/// Monitor enabled work areas
FUNCTION_BLOCK MonitorWorkAreaFB EXTENDS RobotLibraryBaseFB
// ------------------------------------------------------------------------- 
//  SRCI Robot Library                                                
// ------------------------------------------------------------------------- 
//                                                                           
//  Object:      MonitorWorkAreaFB                                       
//  Author:      Thorsten Brach                                                
//  Date:        2024-06-01
//
//  Description:                                              
//   
//                                                                           
//  Copyright: 
//    (C) 2024 Thorsten Brach. All rights reserved                                                                         
//                                                                           
//  Disclaimer:                                                                           
//    This project is provided without any guarantee and can be used for   
//    private and commercial purposes. Any commercial use is at the user’s 
//    own risk and responsibility.
//
// -------------------------------------------------------------------------
VAR_INPUT
  /// Start of the command at the rising edge
  Execute            : BOOL;
  /// Index of robot work area to be monitored
  /// • 0 (default)..254
  WorkAreaNo         : USINT;
END_VAR

VAR_OUTPUT
  /// TRUE, while the following outputs return valid values
  /// ActivationState
  /// MonitoringState
  Valid              : BOOL;
  /// FB is being processed
  Busy               : BOOL;
  /// Command is transferred and confirmed by the RC
  CommandBuffered    : BOOL;  
  /// Receiving of input parameter values has been acknowledged by RC
  ParameterAccepted  : BOOL;
  /// Bits return TRUE when work area defined by Index is active
  ActivationState    : WORD;
  /// Bits return TRUE when violation is reported.
  MonitoringState    : WORD;
END_VAR

                  
                

METHOD PROTECTED OnCall
VAR_IN_OUT
  /// Robot assignment of function
  AxesGroup         : AxesGroup; 
END_VAR
                        
                      
END_METHOD
END_FUNCTION_BLOCK

/// Switch path mode between high and low accuracy
FUNCTION_BLOCK PathAccuracyModeFB EXTENDS RobotLibraryBaseFB
// ------------------------------------------------------------------------- 
//  SRCI Robot Library                                                
// ------------------------------------------------------------------------- 
//                                                                           
//  Object:      PathAccuracyModeFB                                       
//  Author:      Thorsten Brach                                                
//  Date:        2024-06-01
//
//  Description:                                              
//   
//                                                                           
//  Copyright: 
//    (C) 2024 Thorsten Brach. All rights reserved                                                                         
//                                                                           
//  Disclaimer:                                                                           
//    This project is provided without any guarantee and can be used for   
//    private and commercial purposes. Any commercial use is at the user’s 
//    own risk and responsibility.
//
// -------------------------------------------------------------------------
VAR_INPUT
  /// Set TRUE to change RA power state to "Enabled"
  Enable            : BOOL;
END_VAR

VAR_OUTPUT
  /// FB is being processed
  Busy              : BOOL;
  /// Command is transferred and confirmed by the RC
  CommandBuffered   : BOOL;
  /// TRUE while PathAccuracyMode is active
  Enabled           : BOOL;
  /// Receiving of input parameter values has been acknowledged by RC
  ParameterAccepted : BOOL;
END_VAR

                  
                

METHOD PROTECTED OnCall
VAR_IN_OUT
  /// Robot assignment of function
  AxesGroup         : AxesGroup; 
END_VAR
                        
                      
END_METHOD
END_FUNCTION_BLOCK

/// Restart/reboot of the RC.
FUNCTION_BLOCK RestartControllerFB EXTENDS RobotLibraryBaseFB
// ------------------------------------------------------------------------- 
//  SRCI Robot Library                                                
// ------------------------------------------------------------------------- 
//                                                                           
//  Object:      RestartControllerFB                                       
//  Author:      Thorsten Brach                                                
//  Date:        2024-06-01
//
//  Description:                                              
//   
//                                                                           
//  Copyright: 
//    (C) 2024 Thorsten Brach. All rights reserved                                                                         
//                                                                           
//  Disclaimer:                                                                           
//    This project is provided without any guarantee and can be used for   
//    private and commercial purposes. Any commercial use is at the user’s 
//    own risk and responsibility.
//
// -------------------------------------------------------------------------
VAR_INPUT
  /// Start of the command at the rising edge
  Execute         : BOOL;
END_VAR

VAR_OUTPUT
  /// The command has been completed successfully
  Done            : BOOL;
  /// FB is being processed
  Busy            : BOOL;
  /// Command is transferred and confirmed by the RC
  CommandBuffered : BOOL;
  /// TRUE when execution of command has been confirmed by RC and restart is about to be initiated.
  RestartAccepted : BOOL;
END_VAR

                  
                

METHOD PROTECTED OnCall
VAR_IN_OUT
  /// Robot assignment of function
  AxesGroup         : AxesGroup; 
END_VAR
                        
                      
END_METHOD
END_FUNCTION_BLOCK

/// Return to path left during active interrupt
FUNCTION_BLOCK ReturnToPrimaryFB EXTENDS RobotLibraryBaseFB
// ------------------------------------------------------------------------- 
//  SRCI Robot Library                                                
// ------------------------------------------------------------------------- 
//                                                                           
//  Object:      ReturnToPrimaryFB                                       
//  Author:      Thorsten Brach                                                
//  Date:        2024-06-01
//
//  Description:                                              
//   
//                                                                           
//  Copyright: 
//    (C) 2024 Thorsten Brach. All rights reserved                                                                         
//                                                                           
//  Disclaimer:                                                                           
//    This project is provided without any guarantee and can be used for   
//    private and commercial purposes. Any commercial use is at the user’s 
//    own risk and responsibility.
//
// -------------------------------------------------------------------------
VAR_INPUT
  /// Start of the command at the rising edge
  Execute            : BOOL;
  /// Defines target position when function is executed:
  /// • 0: Interrupt position (default) - Returns to position active,  when interrupt was executed
  /// • 1: End position                 - Returns to target position of interrupted segment
  ReturnMode         : BOOL;
  /// TCP velocity in % of nominal velocity
  /// •  <0%: (default) - Use default velocity
  /// •   0%:           - Use internal minimal velocity
  /// • 100%:           - Use maximal reference velocity
  /// See chapter 5.5.7 Robot dynamics
  VelocityRate       : REAL;
  /// Acceleration for movement in % of nominal acceleration
  /// •  <0%: (default) - Use default acceleration
  /// •   0%:           - Use internal minimal acceleration
  /// • 100%:           - Use maximal reference acceleration
  /// See chapter 5.5.7 Robot dynamics
  AccelerationRate   : REAL;
  /// Deceleration for movement in % of nominal deceleration
  /// •  <0%: (default) - Use default deceleration 
  /// •   0%:           - Use internal minimal deceleration
  /// • 100%:           - Use maximal reference deceleration
  /// See chapter 5.5.7 Robot dynamics
  DecelerationRate   : REAL;
  /// Jerk of the movement in % of nominal jerk
  /// •  <0%: (default) - Use default jerk
  /// •   0%:           - Use internal minimal jerk
  /// • 100%:           - Use maximal reference jerk
  /// See chapter 5.5.7 Robot dynamics
  JerkRate           : REAL;
  /// Index of tool
  /// •      0: Flange (default)
  /// • 1..254: Tool frames
  ToolNo             : USINT;
  /// Index of frame
  /// •      0: WCS (default)
  /// • 1..254: User frames
  FrameNo            : USINT;
  /// Parameter is used if it is greater than 0 (default):
  /// Maximum allowed distance between current position and target position according to ReturnMode.
  /// If calculated distance is beyond specified Limit, RC returns an error
  DistanceLimit      : REAL;
  /// Defines type of command movement. One of the optional modes must be supported
  TrajectoryMode     : TrajectoryMode;
  /// Parameter is used if it is greater than 0 (default)
  /// • Velocity input is ignored
  /// • Parameter defines the time for the movement to reach the target position
  /// Error is sent by the RC if the time cannot be kept
  MoveTime           : TIME;
  /// Set TRUE to deactivate comparison of
  /// • ToolData and FrameData
  /// • ToolNo and PrimaryPosToolNo
  /// • FrameNo and PrimaryPosFrameNo
  AllowDifferences   : BOOL;
END_VAR

VAR_OUTPUT
  /// The command has been completed successfully
  Done               : BOOL;
  /// FB is being processed
  Busy               : BOOL;
  /// Command is transferred and confirmed by the RC
  CommandBuffered    : BOOL;
  /// The command takes control of the motion of the according axis group
  Active             : BOOL;
  /// The command was aborted by another command.
  CommandAborted     : BOOL;
  /// TRUE, while command is interrupted during execution and can be continued
  CommandInterrupted : BOOL;
  /// Distance-to-go of the current job.
  /// • -1: No valid value because move command is not yet active (valid values are pending) or not supported by RC
  /// • >0: Actual distance between current and target position
  /// •  0: Target position reached
  RemainingDistance  : REAL;
  /// Percentage of already traversed distance of current job.
  /// If not supported : • -1
  Progress           : REAL;
  /// Tool index of target position of ReturnToPrimary
  /// • 0: Flange
  /// • 1..254: Tool frames
  PrimaryPosToolNo   : USINT;
  /// Frame index of target position of ReturnToPrimary
  /// • 0: WCS
  ///• 1..254: User frames
  PrimaryPosFrameNo  : USINT;
END_VAR

                  
                

METHOD PROTECTED OnCall
VAR_IN_OUT
  /// Robot assignment of function
  AxesGroup         : AxesGroup; 
END_VAR
                        
                      
END_METHOD
END_FUNCTION_BLOCK

/// Transform a defined position in space
FUNCTION_BLOCK ShiftPositionFB EXTENDS RobotLibraryBaseFB
// ------------------------------------------------------------------------- 
//  SRCI Robot Library                                                
// ------------------------------------------------------------------------- 
//                                                                           
//  Object:      ShiftPositionFB                                       
//  Author:      Thorsten Brach                                                
//  Date:        2024-06-01
//
//  Description:                                              
//   
//                                                                           
//  Copyright: 
//    (C) 2024 Thorsten Brach. All rights reserved                                                                         
//                                                                           
//  Disclaimer:                                                                           
//    This project is provided without any guarantee and can be used for   
//    private and commercial purposes. Any commercial use is at the user’s 
//    own risk and responsibility.
//
// -------------------------------------------------------------------------
VAR_INPUT
  /// Start of the command at the rising edge
  Execute                   : BOOL;
  /// Define which method should be used to transform the position:
  Mode                      : TransformMode;
  /// Absolute coordinates of the position that will be transformed in the selected coordinate systems (see input parameter CoordinateSystem).
  Position                  : RobotCartesianPosition;
  /// Defines the reference frame ID to which the "Position" that will be transformed is relative.
  /// • 0: WCS (default)
  /// • 1..254: User frames
  FrameNo                   : USINT;
  /// Defines the reference frame ID to which the "TransformedPosition" should be relative.
  /// • 0: WCS (default)
  /// • 1..254: User frames
  TargetFrameNo             : USINT;
  /// Defines the frame data relevant for the transformation of the "Position". Relates to all "Mode" settings. 
  /// The parameter includes the Frame ID to which the origin of the shifting and rotation is relative and the cartesian position of the origin
  TransformationParameter_1 : FrameData;
  /// Relates to all "Mode" settings. Defines the enabled axis or plane as reference straight line or reference plain for the transformation
  TransformationParameter_2 : ReferenceElement;
  /// Defines the angle of rotation around the defined straight line. 
  /// Related to "Mode" with the setting "Rotate around Straight Line".
  RotationAngle             : REAL;
END_VAR
VAR_OUTPUT
  /// The command has been completed successfully
  Done                      : BOOL;
  /// FB is being processed
  Busy                      : BOOL;
  /// Command is transferred and confirmed by the RC
  CommandBuffered           : BOOL;
  /// Tool index
  TransformedPosition       : RobotCartesianPosition;
END_VAR

                  
                

METHOD PROTECTED OnCall
VAR_IN_OUT
  /// Robot assignment of function
  AxesGroup         : AxesGroup; 
END_VAR
                        
                      
END_METHOD
END_FUNCTION_BLOCK

/// Push robot: Robot calculates opposite vector and moves slowly in that direction
FUNCTION_BLOCK SoftSwitchTcpFB EXTENDS RobotLibraryBaseFB
// ------------------------------------------------------------------------- 
//  SRCI Robot Library                                                
// ------------------------------------------------------------------------- 
//                                                                           
//  Object:      SoftSwitchTcpFB                                       
//  Author:      Thorsten Brach                                                
//  Date:        2024-06-01
//
//  Description:                                              
//   
//                                                                           
//  Copyright: 
//    (C) 2024 Thorsten Brach. All rights reserved                                                                         
//                                                                           
//  Disclaimer:                                                                           
//    This project is provided without any guarantee and can be used for   
//    private and commercial purposes. Any commercial use is at the user’s 
//    own risk and responsibility.
//
// -------------------------------------------------------------------------
VAR_INPUT
  /// Start of the command at the rising edge
  Execute             : BOOL;
  /// Defines type of reference coordinate system at which the robot can be moved in a compliant manner.
  ReferenceType       : ReferenceType;
  /// Index of tool or frame according to ReferenceType.
  /// • 0 (default): Flange/WS
  /// • 1..254: Tool/User frames
  ReferenceNo         : USINT;
  /// Parameter which determines the behavior towards the previously sent and still active or buffered commands
  AbortingMode        : AbortingMode;
  /// Relates to "LimitMode" with the setting "No limit defined". Defines for which cartesian axes the compliant motion is allowed. 
  /// If TRUE, the direction is enabled. Default value is FALSE. See Table 6-744 for bit assignment.
  CompliantAxes       : BYTE;
  /// Defines which parameters will limit the space, where the robot complies (at least one option must be supported)
  LimitMode           : LimitMode;
  /// Defines the type of the resistance force applied at the RA against the external force
  ResistanceForceMode : ResistanceForceMode;
  /// Relates to "ResistanceForceMode" with the setting "ResistanceForceTCP".
  /// Defines the resistance force level applied at the RA against the external force.
  /// • 0..99: Resistance is lower than robot vendor default. The lower the value, the easier the robot can be pushed away.
  /// • 100 (default): The value is aligned with the robot vendor-specific default value.
  /// • 101..200: Resistance is higher than robot vendor default. At maximum value "200" highest possible resistance against external force
  ResistanceForceTCP  : REAL;
  /// Relates to "ResistanceForceMode" with the setting "ResistanceForceAxis".
  /// Defines the resistance force level of the RA at the respective cartesian axis.
  ///  0..99: Resistance is lower than robot vendor default. The lower the value, the easier the robot can be pushed away.
  /// • 100 (default): The value is aligned with the robot vendor-specific default value.
  /// • 101..200: Resistance is higher than robot vendor default. At maximum value "200" highest possible resistance against external force.
  /// Index:
  /// • [0]: X-Axis O
  /// • [1]: Y-axis O
  /// • [2]: Z-axis O
  /// • [3]: RX-Direction O
  /// • [4]: RY-direction O
  /// • [5]: RZ-direction
  ResistanceForceAxis : ARRAY[0..5] OF REAL;
  /// Relates to "LimitMode" with the setting "Limit defined". 
  /// Limit values in the selected cartesian coordinate system (see input parameters ReferenceType and ReferenceNo).
  /// "0" is (default) the origin of the vector, the TCP position, at the start position of the robot.
  /// See Table 6-742 for the parameter index assignment.
  VectorData          : ARRAY[0..5] OF REAL;
  /// Defines the target sequence in which the command will be executed
  SequenceFlag        : SequenceFlag;
END_VAR
VAR_OUTPUT
  /// The command has been completed successfully
  Done                : BOOL;
  /// FB is being processed
  Busy                : BOOL;
  /// Command is transferred and confirmed by the RC
  CommandBuffered     : BOOL;
  /// The command "SoftSwitchTCP" takes control of the according axis group.
  Active              : BOOL;
  /// The command was aborted by another command
  CommandAborted      : BOOL;
  /// TRUE, while command is interrupted during execution and can be continued
  CommandInterrupted  : BOOL;
  /// If TRUE, the RA is in a compliant movement.
  SoftMovement        : BOOL;
END_VAR

                  
                

METHOD PROTECTED OnCall
VAR_IN_OUT
  /// Robot assignment of function
  AxesGroup         : AxesGroup; 
END_VAR
                        
                      
END_METHOD
END_FUNCTION_BLOCK

/// Switch language of robot teach pendant from PLC
FUNCTION_BLOCK SwitchLanguageFB EXTENDS RobotLibraryBaseFB
// ------------------------------------------------------------------------- 
//  SRCI Robot Library                                                
// ------------------------------------------------------------------------- 
//                                                                           
//  Object:      SwitchLanguageFB                                       
//  Author:      Thorsten Brach                                                
//  Date:        2024-06-01
//
//  Description:                                              
//   
//                                                                           
//  Copyright: 
//    (C) 2024 Thorsten Brach. All rights reserved                                                                         
//                                                                           
//  Disclaimer:                                                                           
//    This project is provided without any guarantee and can be used for   
//    private and commercial purposes. Any commercial use is at the user’s 
//    own risk and responsibility.
//
// -------------------------------------------------------------------------
VAR_INPUT
  /// Start of the command at the rising edge
  Execute            : BOOL;
  /// Two letter code of language to be set at the original operating panel of the robot (default: EN)
  LanguageCode       : STRING(2);
END_VAR


VAR_OUTPUT
  /// The command has been completed successfully
  Done               : BOOL;
  /// FB is being processed
  Busy               : BOOL;
  /// Command is transferred and confirmed by the RC
  CommandBuffered    : BOOL;
  /// Two letter code of actual language used at the original operating panel of the robot.
  ActualLanguageCode : STRING(2);
END_VAR

                  
                

METHOD PROTECTED OnCall
VAR_IN_OUT
  /// Robot assignment of function
  AxesGroup         : AxesGroup; 
END_VAR
                        
                      
END_METHOD
END_FUNCTION_BLOCK

/// Measure the length of objects in the cartesian space, execution time for specified section of a job or signal output time of a specified signal
FUNCTION_BLOCK UnitMeasurementFB EXTENDS RobotLibraryBaseFB
// ------------------------------------------------------------------------- 
//  SRCI Robot Library                                                
// ------------------------------------------------------------------------- 
//                                                                           
//  Object:      UnitMeasurementFB                                       
//  Author:      Thorsten Brach                                                
//  Date:        2024-06-01
//
//  Description:                                              
//   
//                                                                           
//  Copyright: 
//    (C) 2024 Thorsten Brach. All rights reserved                                                                         
//                                                                           
//  Disclaimer:                                                                           
//    This project is provided without any guarantee and can be used for   
//    private and commercial purposes. Any commercial use is at the user’s 
//    own risk and responsibility.
//
// -------------------------------------------------------------------------
VAR_INPUT
  /// Set TRUE to activate "UnitMeasurement".
  Enable            : BOOL;
  ///  Reaction type of measurement in relation to the trigger signal with the "ListenerID > 0" (at least one option must be supported):
  TriggerMode       : TriggerModeMeasurement;
  /// Relates to "TriggerMode" "No trigger related behavior".
  /// Set TRUE to start first measurement. Set TRUE again to receive new result data referring to previous rising edge of NewMeasurement.
  NewMeasurement    : BOOL;
  /// Type of measurement (at least one option must be supported). 
 /// If the parameter is changed during the active measurement, the RC returns an error
  MeasuringMode     : MeasuringUnitMode;
  /// ID of the trigger function that may be triggered:
  /// • 0: Immediately (default). - Start executing THIS function immediately.
  /// • >0: Triggero Start executing when the trigger function with the identical EmitterID is called.
  /// For more information see chapter 5.5.12.4.
  ListenerID         : SINT;


END_VAR

VAR_OUTPUT
  /// FB is being processed
  Busy              : BOOL;
  /// Command is transferred and confirmed by the RC
  CommandBuffered   : BOOL;
  /// TRUE while "FreeDrive" is active.
  Enabled           : BOOL;
  /// Receiving of input parameter values has been acknowledged by RC
  ParameterAccepted : BOOL;
  /// TRUE, while the measurement is active.
  MeasurementActive : BOOL;
  /// Measurement result depending on the measurement type setting of the "MeasuringMode".
  Result            : REAL;
  /// Unique system-generated ID of the "Action" when the function is triggered.
  /// • >0: The "Action" is started by the trigger function with identical FollowID.
  /// • <0: The "Action" is stopped by the trigger function with identical FollowID.
  /// For more information see chapter 5.5.12.4 EmitterID, ListenerID, FollowID and OriginID
  OriginID           : INT;
  /// Relates to ListenerID >0
  /// Number of successful trigger -based command invocations
  /// For more information refer to chapter 5.5.12.4.
  InvocationCounter  : USINT;
END_VAR

                  
                

METHOD PROTECTED OnCall
VAR_IN_OUT
  /// Robot assignment of function
  AxesGroup         : AxesGroup; 
END_VAR
                        
                      
END_METHOD
END_FUNCTION_BLOCK

/// Login on RC from PLC
FUNCTION_BLOCK UserLoginFB EXTENDS RobotLibraryBaseFB
// ------------------------------------------------------------------------- 
//  SRCI Robot Library                                                
// ------------------------------------------------------------------------- 
//                                                                           
//  Object:      UserLoginFB                                       
//  Author:      Thorsten Brach                                                
//  Date:        2024-06-01
//
//  Description:                                              
//   
//                                                                           
//  Copyright: 
//    (C) 2024 Thorsten Brach. All rights reserved                                                                         
//                                                                           
//  Disclaimer:                                                                           
//    This project is provided without any guarantee and can be used for   
//    private and commercial purposes. Any commercial use is at the user’s 
//    own risk and responsibility.
//
// -------------------------------------------------------------------------
VAR_INPUT
  /// Start of the command at the rising edge
  Execute         : BOOL;
  /// Defines the logon type (at least one option must be supported)
  Mode            : LogonMode;
  /// Defines the user password.
  Password        : STRING(50);
  /// Defines the name of the operator
  Username        : STRING(50);
  /// Defines the level ID of the operator (default: 0)
  LevelID         : SINT;
END_VAR
VAR_OUTPUT
  /// The command has been completed successfully
  Done            : BOOL;
  /// FB is being processed
  Busy            : BOOL;
  /// Command is transferred and confirmed by the RC
  CommandBuffered : BOOL;
END_VAR

                  
                

METHOD PROTECTED OnCall
VAR_IN_OUT
  /// Robot assignment of function
  AxesGroup         : AxesGroup; 
END_VAR
                        
                      
END_METHOD
END_FUNCTION_BLOCK

/// Set wait command between motion commands
FUNCTION_BLOCK WaitTimeFB EXTENDS RobotLibraryBaseFB
// ------------------------------------------------------------------------- 
//  SRCI Robot Library                                                
// ------------------------------------------------------------------------- 
//                                                                           
//  Object:      WaitTimeFB                                       
//  Author:      Thorsten Brach                                                
//  Date:        2024-06-01
//
//  Description:                                              
//   
//                                                                           
//  Copyright: 
//    (C) 2024 Thorsten Brach. All rights reserved                                                                         
//                                                                           
//  Disclaimer:                                                                           
//    This project is provided without any guarantee and can be used for   
//    private and commercial purposes. Any commercial use is at the user’s 
//    own risk and responsibility.
//
// -------------------------------------------------------------------------
VAR_INPUT
  /// Start of the command at the rising edge
  Execute            : BOOL;
  /// Parameter which determines the behavior towards the previously sent and still active or buffered commands
  AbortingMode       : AbortingMode;
  /// Duration [ms] of the waiting time. The value of the parameter must be positive
  WaitTime           : UDINT;
  /// Defines the target sequence in which the command will be executed
  SequenceFlag       : SequenceFlag;
END_VAR
VAR_OUTPUT
  /// The command has been completed successfully
  Done               : BOOL;
  /// FB is being processed
  Busy               : BOOL;
  /// Command is transferred and confirmed by the RC
  CommandBuffered    : BOOL;
  /// Command is currently processed by the active sequence, takes control of the motion of the
  /// according axis group and is waiting for the time specified via "Time" to elapse.
  Active             : BOOL;
  /// The command was aborted by another command.
  CommandAborted     : BOOL;
  /// TRUE, while command is interrupted during execution and can be continued.
  CommandInterrupted : BOOL;
  /// Current value of time [ms] that has elapsed since processing of the command has started.
  ElapsedTime        : UDINT;
END_VAR

                  
                

METHOD PROTECTED OnCall
VAR_IN_OUT
  /// Robot assignment of function
  AxesGroup         : AxesGroup; 
END_VAR
                        
                      
END_METHOD
END_FUNCTION_BLOCK

/// Direct Move to target position through auxiliary position defined
/// by offset in all dimensions (movement to target posi tion PTP)
FUNCTION_BLOCK MoveApproachDirectFB EXTENDS RobotLibraryBaseFB
// ------------------------------------------------------------------------- 
//  SRCI Robot Library                                                
// ------------------------------------------------------------------------- 
//                                                                           
//  Object:      MoveApproachDirectFB                                       
//  Author:      Thorsten Brach                                                
//  Date:        2024-06-01
//
//  Description:                                              
//   
//                                                                           
//  Copyright: 
//    (C) 2024 Thorsten Brach. All rights reserved                                                                         
//                                                                           
//  Disclaimer:                                                                           
//    This project is provided without any guarantee and can be used for   
//    private and commercial purposes. Any commercial use is at the user’s 
//    own risk and responsibility.
//
// -------------------------------------------------------------------------
VAR_INPUT
  /// Start of the command at the rising edge
  Execute            : BOOL;
  /// Absolute target coordinates in the selected coordinate system (see input parameters ToolNo and FrameNo).
  TargetPosition     : RobotCartesianPosition;
  /// Offset distance of auxiliary position from TargetPosition
  Offset             : AuxOffset;
  /// Defines type of reference coordinate system of the offset position
  ReferenceType      : ReferenceType;
  /// TCP velocity in % of nominal velocity
  /// •  <0%: (default) - Use default velocity
  /// •   0%:           - Use internal minimal velocity
  /// • 100%:           - Use maximal reference velocity
  /// See chapter 5.5.7 Robot dynamics
  VelocityRate       : REAL;
  /// Acceleration for movement in % of nominal acceleration
  /// •  <0%: (default) - Use default acceleration
  /// •   0%:           - Use internal minimal acceleration
  /// • 100%:           - Use maximal reference acceleration
  /// See chapter 5.5.7 Robot dynamics
  AccelerationRate   : REAL;
  /// Deceleration for movement in % of nominal deceleration
  /// •  <0%: (default) - Use default deceleration 
  /// •   0%:           - Use internal minimal deceleration
  /// • 100%:           - Use maximal reference deceleration
  /// See chapter 5.5.7 Robot dynamics
  DecelerationRate   : REAL;
  /// Jerk of the movement in % of nominal jerk
  /// •  <0%: (default) - Use default jerk
  /// •   0%:           - Use internal minimal jerk
  /// • 100%:           - Use maximal reference jerk
  /// See chapter 5.5.7 Robot dynamics
  JerkRate           : REAL;
  /// Index of tool
  /// •      0: Flange (default)
  /// • 1..254: Tool frames
  ToolNo             : USINT;
  /// Index of frame
  /// •      0: WCS (default)
  /// • 1..254: User frames
  FrameNo            : USINT;
  /// Parameter which determines the behavior towards the previously sent and still active or buffered commands
  AbortingMode       : AbortingMode;
  /// Parameter which determines the transition behavior at the end of the movement to be sent to the next command. 
  /// The user can choose a transition type between exact stop and different blend possibilities
  BlendingMode       : BlendingMode;
  /// Additional parameter for the blending mode, to define i.e. velocity limit (%) or blending radius
  BlendingParameter  : ARRAY [0..1] OF REAL := [10,0];
  /// Define blending sphere with radius around auxiliary position. For exact stop define AuxCornerDistance = 0
  AuxCornerDistance  : REAL;
  /// Parameter is used if it is greater than 0 (default)
  /// • Velocity input is ignored
  /// • Parameter defines the time for the movement to reach the target position
  /// Error is sent by the RC if the time cannot be kept
  MoveTime           : TIME;
  /// Parameter to describe how the orientation axes (RX, RY, RZ) will be interpolated during the movement
  OriMode            : OriMode;
  /// Defines the usage of the config byte inside the position according to Table 6-238
  ConfigMode         : ArmConfigParameter;
  /// Defines the usage of the TurnNumber byte inside the position.
  TurnMode           : TurnMode;
  /// Factor by which VelocityRate is multiplied to define the velocity for the second segment of the motion. Always positive.
  /// • 0: use the minimal velocity
  /// • 1: use the velocity set with VelocityRate 
  /// Input values below 1 to reduce velocity, 
  /// Input values above 1 to increase velocity.
  /// See chapter 5.5.7 Robot dynamics
  VelocityCoefficient: REAL;
  /// Set TRUE to allow manipulation of this move command through superimposing functions.
  /// For more information see chapter 5.5.9.5
  Manipulation       : BOOL;
  /// Defines the target sequence in which the command will be executed
  SequenceFlag       : SequenceFlag;
  /// ID of Action that will be executed when this command is active
  /// • >0: Start Action - Start executing the Action function with the identical ListenerID.
  /// • <0: Stop Action  -  Stop executing the Action function with the identical ListenerID.
  /// • 0: No trigger (default)-  If no EmitterID is defined, the function will not trigger any Action during its execution
  /// For more information see section Triggers of this chapter or chapter 5.5.12.4.
  EmitterID          : ARRAY [0..3] OF SINT;
END_VAR

VAR_OUTPUT
  /// The command has been completed successfully
  Done               : BOOL;
  /// FB is being processed
  Busy               : BOOL;
  /// Command is transferred and confirmed by the RC
  CommandBuffered    : BOOL;
  /// The command takes control of the motion of the according axis group
  Active             : BOOL;
  /// The command was aborted by another command.
  CommandAborted     : BOOL;
  /// TRUE, while command is interrupted during execution and can be continued
  CommandInterrupted : BOOL;
  /// Distance-to-go of the current job.
  /// • -1: No valid value because move command is not yet active (valid values are pending) or not supported by RC
  /// • >0: Actual distance between current and target position
  /// •  0: Target position reached
  RemainingDistance  : REAL;
  /// Percentage of already traversed distance of current job.
  /// If not supported : • -1
  Progress           : REAL;
  /// Unique system-generated ID of the trigger function when the function is called by the user.
  /// For more information see chapter 5.5.12.4.
  FollowID           : DINT;
END_VAR

                  
                

METHOD PROTECTED OnCall
VAR_IN_OUT
  /// Robot assignment of function
  AxesGroup         : AxesGroup; 
END_VAR
                        
                      
END_METHOD
END_FUNCTION_BLOCK

/// Linear Move to target position through auxiliary position defined by offset in all dimensions (movement to target position linear)
FUNCTION_BLOCK MoveApproachLinearFB EXTENDS RobotLibraryBaseFB
// ------------------------------------------------------------------------- 
//  SRCI Robot Library                                                
// ------------------------------------------------------------------------- 
//                                                                           
//  Object:      MoveApproachLinearFB                                       
//  Author:      Thorsten Brach                                                
//  Date:        2024-06-01
//
//  Description:                                              
//   
//                                                                           
//  Copyright: 
//    (C) 2024 Thorsten Brach. All rights reserved                                                                         
//                                                                           
//  Disclaimer:                                                                           
//    This project is provided without any guarantee and can be used for   
//    private and commercial purposes. Any commercial use is at the user’s 
//    own risk and responsibility.
//
// -------------------------------------------------------------------------
VAR_INPUT
  /// Start of the command at the rising edge
  Execute            : BOOL;
  /// Absolute target coordinates in the selected coordinate system (see input parameters ToolNo and FrameNo).
  TargetPosition     : RobotCartesianPosition;
  /// Offset distance of auxiliary position from TargetPosition
  Offset             : AuxOffset;
  /// Defines type of reference coordinate system of the offset position
  ReferenceType      : ReferenceType;
  /// TCP velocity in % of nominal velocity
  /// •  <0%: (default) - Use default velocity
  /// •   0%:           - Use internal minimal velocity
  /// • 100%:           - Use maximal reference velocity
  /// See chapter 5.5.7 Robot dynamics
  VelocityRate       : REAL;
  /// Acceleration for movement in % of nominal acceleration
  /// •  <0%: (default) - Use default acceleration
  /// •   0%:           - Use internal minimal acceleration
  /// • 100%:           - Use maximal reference acceleration
  /// See chapter 5.5.7 Robot dynamics
  AccelerationRate   : REAL;
  /// Deceleration for movement in % of nominal deceleration
  /// •  <0%: (default) - Use default deceleration 
  /// •   0%:           - Use internal minimal deceleration
  /// • 100%:           - Use maximal reference deceleration
  /// See chapter 5.5.7 Robot dynamics
  DecelerationRate   : REAL;
  /// Jerk of the movement in % of nominal jerk
  /// •  <0%: (default) - Use default jerk
  /// •   0%:           - Use internal minimal jerk
  /// • 100%:           - Use maximal reference jerk
  /// See chapter 5.5.7 Robot dynamics
  JerkRate           : REAL;
  /// Index of tool
  /// •      0: Flange (default)
  /// • 1..254: Tool frames
  ToolNo             : USINT;
  /// Index of frame
  /// •      0: WCS (default)
  /// • 1..254: User frames
  FrameNo            : USINT;
  /// Parameter which determines the behavior towards the previously sent and still active or buffered commands
  AbortingMode       : AbortingMode;
  /// Parameter which determines the transition behavior at the end of the movement to be sent to the next command. 
  /// The user can choose a transition type between exact stop and different blend possibilities
  BlendingMode       : BlendingMode;
  /// Additional parameter for the blending mode, to define i.e. velocity limit (%) or blending radius
  BlendingParameter  : ARRAY [0..1] OF REAL := [10,0];
  /// Define blending sphere with radius around auxiliary position. For exact stop define AuxCornerDistance = 0
  AuxCornerDistance  : REAL;
  /// Parameter is used if it is greater than 0 (default)
  /// • Velocity input is ignored
  /// • Parameter defines the time for the movement to reach the target position
  /// Error is sent by the RC if the time cannot be kept
  MoveTime           : TIME;
  /// Parameter to describe how the orientation axes (RX, RY, RZ) will be interpolated during the movement
  OriMode            : OriMode;
  /// Defines the usage of the config byte inside the position according to Table 6-238
  ConfigMode         : ArmConfigParameter;
  /// Defines the usage of the TurnNumber byte inside the position.
  TurnMode           : TurnMode;
  /// Factor by which VelocityRate is multiplied to define the velocity for the second segment of the motion. Always positive.
  /// • 0: use the minimal velocity
  /// • 1: use the velocity set with VelocityRate 
  /// Input values below 1 to reduce velocity, 
  /// Input values above 1 to increase velocity.
  /// See chapter 5.5.7 Robot dynamics
  VelocityCoefficient: REAL;
  /// Set TRUE to allow manipulation of this move command through superimposing functions.
  /// For more information see chapter 5.5.9.5
  Manipulation       : BOOL;
  /// Defines the target sequence in which the command will be executed
  SequenceFlag       : SequenceFlag;
  /// ID of Action that will be executed when this command is active
  /// • >0: Start Action - Start executing the Action function with the identical ListenerID.
  /// • <0: Stop Action  -  Stop executing the Action function with the identical ListenerID.
  /// • 0: No trigger (default)-  If no EmitterID is defined, the function will not trigger any Action during its execution
  /// For more information see section Triggers of this chapter or chapter 5.5.12.4.
  EmitterID          : ARRAY [0..3] OF SINT;
END_VAR

VAR_OUTPUT
  /// The command has been completed successfully
  Done               : BOOL;
  /// FB is being processed
  Busy               : BOOL;
  /// Command is transferred and confirmed by the RC
  CommandBuffered    : BOOL;
  /// The command takes control of the motion of the according axis group
  Active             : BOOL;
  /// The command was aborted by another command.
  CommandAborted     : BOOL;
  /// TRUE, while command is interrupted during execution and can be continued
  CommandInterrupted : BOOL;
  /// Distance-to-go of the current job.
  /// • -1: No valid value because move command is not yet active (valid values are pending) or not supported by RC
  /// • >0: Actual distance between current and target position
  /// •  0: Target position reached
  RemainingDistance  : REAL;
  /// Percentage of already traversed distance of current job.
  /// If not supported : • -1
  Progress           : REAL;
  /// Unique system-generated ID of the trigger function when the function is called by the user.
  /// For more information see chapter 5.5.12.4.
  FollowID           : DINT;
END_VAR

                  
                

METHOD PROTECTED OnCall
VAR_IN_OUT
  /// Robot assignment of function
  AxesGroup         : AxesGroup; 
END_VAR
                        
                      
END_METHOD
END_FUNCTION_BLOCK

/// Move all joints to an absolute joint position (Absolute Joint PTP)
FUNCTION_BLOCK MoveAxesAbsoluteFB EXTENDS RobotLibraryBaseFB
// ------------------------------------------------------------------------- 
//  SRCI Robot Library                                                
// ------------------------------------------------------------------------- 
//                                                                           
//  Object:      MoveAxesAbsoluteFB                                       
//  Author:      Thorsten Brach                                                
//  Date:        2024-06-01
//
//  Description:                                              
//   
//                                                                           
//  Copyright: 
//    (C) 2024 Thorsten Brach. All rights reserved                                                                         
//                                                                           
//  Disclaimer:                                                                           
//    This project is provided without any guarantee and can be used for   
//    private and commercial purposes. Any commercial use is at the user’s 
//    own risk and responsibility.
//
// -------------------------------------------------------------------------
VAR_INPUT
  /// Start of the command at the rising edge
  Execute            : BOOL;
  /// Absolute end position of the robot in Joint position.
  JointPosition      : RobotJointPosition;
  /// Axes velocity in % of nominal velocity.
  /// •  <0%: (default) - Use default velocity
  /// •   0%:           - Use internal minimal velocity
  /// • 100%:           - Use maximal reference velocity
  /// See chapter 5.5.7 Robot dynamics
  VelocityRate       : REAL;
  /// Acceleration for movement in % of nominal acceleration
  /// •  <0%: (default) - Use default acceleration
  /// •   0%:           - Use internal minimal acceleration
  /// • 100%:           - Use maximal reference acceleration
  /// See chapter 5.5.7 Robot dynamics
  AccelerationRate   : REAL;
  /// Deceleration for movement in % of nominal deceleration
  /// •  <0%: (default) - Use default deceleration 
  /// •   0%:           - Use internal minimal deceleration
  /// • 100%:           - Use maximal reference deceleration
  /// See chapter 5.5.7 Robot dynamics
  DecelerationRate   : REAL;
  /// Jerk of the movement in % of nominal jerk
  /// •  <0%: (default) - Use default jerk
  /// •   0%:           - Use internal minimal jerk
  /// • 100%:           - Use maximal reference jerk
  /// See chapter 5.5.7 Robot dynamics
  JerkRate           : REAL;
  /// Index of tool
  /// •      0: Flange (default)
  /// • 1..254: Tool frames
  ToolNo             : USINT;
  /// Parameter which determines the behavior towards the previously sent and still active or buffered commands
  AbortingMode       : AbortingMode;
  /// Parameter which determines the transition behavior at the end of the movement to be sent to the next command. 
  /// The user can choose a transition type between exact stop and different blend possibilities
  BlendingMode       : BlendingMode;
  /// Additional parameter for the blending mode, to define i.e. velocity limit (%) or blending radius
  BlendingParameter  : ARRAY [0..1] OF REAL := [10,0];
  /// Parameter is used if it is greater than 0 (default)
  /// • Velocity input is ignored
  /// • Parameter defines the time for the movement to reach the target position
  /// Error is sent by the RC if the time cannot be kept
  MoveTime           : TIME;
  /// Defines the usage of the config byte inside the position according to Table 6-238
  ConfigMode         : ArmConfigParameter;
  /// Set TRUE to allow manipulation of this move command through superimposing functions.
  /// For more information see chapter 5.5.9.5
  Manipulation       : BOOL;
  /// Defines the target sequence in which the command will be executed
  SequenceFlag       : SequenceFlag;
  /// ID of Action that will be executed when this command is active
  /// • >0: Start Action - Start executing the Action function with the identical ListenerID.
  /// • <0: Stop Action  -  Stop executing the Action function with the identical ListenerID.
  /// • 0: No trigger (default)-  If no EmitterID is defined, the function will not trigger any Action during its execution
  /// For more information see section Triggers of this chapter or chapter 5.5.12.4.
  EmitterID          : ARRAY [0..3] OF SINT;
END_VAR

VAR_OUTPUT
  /// The command has been completed successfully
  Done               : BOOL;
  /// FB is being processed
  Busy               : BOOL;
  /// Command is transferred and confirmed by the RC
  CommandBuffered    : BOOL;
  /// The command takes control of the motion of the according axis group
  Active             : BOOL;
  /// The command was aborted by another command.
  CommandAborted     : BOOL;
  /// TRUE, while command is interrupted during execution and can be continued
  CommandInterrupted : BOOL;
  /// Percentage of already traversed distance of current job.
  /// If not supported : • -1
  Progress           : REAL;
  /// Unique system-generated ID of the trigger function when the function is called by the user.
  /// For more information see chapter 5.5.12.4.
  FollowID           : DINT;
END_VAR

                  
                

METHOD PROTECTED OnCall
VAR_IN_OUT
  /// Robot assignment of function
  AxesGroup         : AxesGroup; 
END_VAR
                        
                      
END_METHOD
END_FUNCTION_BLOCK

/// Move all joints relative to actual joint position (Relative Joint PTP)
FUNCTION_BLOCK MoveAxesRelativeFB EXTENDS RobotLibraryBaseFB
// ------------------------------------------------------------------------- 
//  SRCI Robot Library                                                
// ------------------------------------------------------------------------- 
//                                                                           
//  Object:      MoveAxesRelativeFB                                       
//  Author:      Thorsten Brach                                                
//  Date:        2024-06-01
//
//  Description:                                              
//   
//                                                                           
//  Copyright: 
//    (C) 2024 Thorsten Brach. All rights reserved                                                                         
//                                                                           
//  Disclaimer:                                                                           
//    This project is provided without any guarantee and can be used for   
//    private and commercial purposes. Any commercial use is at the user’s 
//    own risk and responsibility.
//
// -------------------------------------------------------------------------
VAR_INPUT
  /// Start of the command at the rising edge
  Execute            : BOOL;
  /// Relative joint distance from the current or last target position to the end joint position
  JointDistance      : RobotJointPosition;
  /// Axes velocity in % of nominal velocity.
  /// •  <0%: (default) - Use default velocity
  /// •   0%:           - Use internal minimal velocity
  /// • 100%:           - Use maximal reference velocity
  /// See chapter 5.5.7 Robot dynamics
  VelocityRate       : REAL;
  /// Acceleration for movement in % of nominal acceleration
  /// •  <0%: (default) - Use default acceleration
  /// •   0%:           - Use internal minimal acceleration
  /// • 100%:           - Use maximal reference acceleration
  /// See chapter 5.5.7 Robot dynamics
  AccelerationRate   : REAL;
  /// Deceleration for movement in % of nominal deceleration
  /// •  <0%: (default) - Use default deceleration 
  /// •   0%:           - Use internal minimal deceleration
  /// • 100%:           - Use maximal reference deceleration
  /// See chapter 5.5.7 Robot dynamics
  DecelerationRate   : REAL;
  /// Jerk of the movement in % of nominal jerk
  /// •  <0%: (default) - Use default jerk
  /// •   0%:           - Use internal minimal jerk
  /// • 100%:           - Use maximal reference jerk
  /// See chapter 5.5.7 Robot dynamics
  JerkRate           : REAL;
  /// Index of tool
  /// •      0: Flange (default)
  /// • 1..254: Tool frames
  ToolNo             : USINT;
  /// Parameter which determines the behavior towards the previously sent and still active or buffered commands
  AbortingMode       : AbortingMode;
  /// Parameter which determines the transition behavior at the end of the movement to be sent to the next command. 
  /// The user can choose a transition type between exact stop and different blend possibilities
  BlendingMode       : BlendingMode;
  /// Additional parameter for the blending mode, to define i.e. velocity limit (%) or blending radius
  BlendingParameter  : ARRAY [0..1] OF REAL := [10,0];
  /// Parameter is used if it is greater than 0 (default)
  /// • Velocity input is ignored
  /// • Parameter defines the time for the movement to reach the target position
  /// Error is sent by the RC if the time cannot be kept
  MoveTime           : TIME;
  /// Set TRUE to allow manipulation of this move command through superimposing functions.
  /// For more information see chapter 5.5.9.5
  Manipulation       : BOOL;
  /// Defines the target sequence in which the command will be executed
  SequenceFlag       : SequenceFlag;
  /// ID of Action that will be executed when this command is active
  /// • >0: Start Action - Start executing the Action function with the identical ListenerID.
  /// • <0: Stop Action  -  Stop executing the Action function with the identical ListenerID.
  /// • 0: No trigger (default)-  If no EmitterID is defined, the function will not trigger any Action during its execution
  /// For more information see section Triggers of this chapter or chapter 5.5.12.4.
  EmitterID          : ARRAY [0..3] OF SINT;
END_VAR

VAR_OUTPUT
  /// The command has been completed successfully
  Done               : BOOL;
  /// FB is being processed
  Busy               : BOOL;
  /// Command is transferred and confirmed by the RC
  CommandBuffered    : BOOL;
  /// The command takes control of the motion of the according axis group
  Active             : BOOL;
  /// The command was aborted by another command.
  CommandAborted     : BOOL;
  /// TRUE, while command is interrupted during execution and can be continued
  CommandInterrupted : BOOL;
  /// Percentage of already traversed distance of current job.
  /// If not supported : • -1
  Progress           : REAL;
  /// Unique system-generated ID of the trigger function when the function is called by the user.
  /// For more information see chapter 5.5.12.4.
  FollowID           : DINT;
END_VAR

                  
                

METHOD PROTECTED OnCall
VAR_IN_OUT
  /// Robot assignment of function
  AxesGroup         : AxesGroup; 
END_VAR
                        
                      
END_METHOD
END_FUNCTION_BLOCK

/// Move the TCP to an absolute cartesian position (circular interpolation)
FUNCTION_BLOCK MoveCircularAbsoluteFB EXTENDS RobotLibraryBaseFB
// ------------------------------------------------------------------------- 
//  SRCI Robot Library                                                
// ------------------------------------------------------------------------- 
//                                                                           
//  Object:      MoveCircularAbsoluteFB                                       
//  Author:      Thorsten Brach                                                
//  Date:        2024-06-01
//
//  Description:                                              
//   
//                                                                           
//  Copyright: 
//    (C) 2024 Thorsten Brach. All rights reserved                                                                         
//                                                                           
//  Disclaimer:                                                                           
//    This project is provided without any guarantee and can be used for   
//    private and commercial purposes. Any commercial use is at the user’s 
//    own risk and responsibility.
//
// -------------------------------------------------------------------------
VAR_INPUT
  /// Start of the command at the rising edge
  Execute            : BOOL;
  /// Specifies the meaning of the input parameter "AuxPoint".
  CircMode           : CircMode;
  /// Auxiliary position of the robot in the specified coordinate system, used in for the circle path calculation.
  AuxPoint           : RobotCartesianPosition;
  /// Specifies the circle’s plane when CircMode = 2 is selected
  CircPlane          : CircPlane;
  /// Relates to CircMode =1:
  /// Permissible deviation of the distances from starting point to center point, from auxiliary point to center point and from end point to center point.
  /// These distances must be identical to travel a circular path. When the distance from a point to the center point is within the allowed deviation, 
  /// the position of the center point is adjusted to the mean internally. If the deviation is greater than the specified Tolerance, 
  /// the command returns an error. See also Figure 6-106.
  Tolerance          : REAL;
  /// Absolute end position of the robot in the specified coordinate system. If "CircMode" = 2 this position is ignored 
  EndPoint           : RobotCartesianPosition;
  /// Angle is only used when "CircMode" = 2. 
  /// The circular angle defines the end position of the circular motion. The circular path is defined by the angle, 
  /// the center point ("AuxPoint") and the actual position. Always positive
  Angle              : REAL;
  /// Choice of the path
  PathChoice         : PathChoice;  
  /// TCP velocity in % of nominal velocity
  /// •  <0%: (default) - Use default velocity
  /// •   0%:           - Use internal minimal velocity
  /// • 100%:           - Use maximal reference velocity
  /// See chapter 5.5.7 Robot dynamics
  VelocityRate       : REAL;
  /// Acceleration for movement in % of nominal acceleration
  /// •  <0%: (default) - Use default acceleration
  /// •   0%:           - Use internal minimal acceleration
  /// • 100%:           - Use maximal reference acceleration
  /// See chapter 5.5.7 Robot dynamics
  AccelerationRate   : REAL;
  /// Deceleration for movement in % of nominal deceleration
  /// •  <0%: (default) - Use default deceleration 
  /// •   0%:           - Use internal minimal deceleration
  /// • 100%:           - Use maximal reference deceleration
  /// See chapter 5.5.7 Robot dynamics
  DecelerationRate   : REAL;
  /// Jerk of the movement in % of nominal jerk
  /// •  <0%: (default) - Use default jerk
  /// •   0%:           - Use internal minimal jerk
  /// • 100%:           - Use maximal reference jerk
  /// See chapter 5.5.7 Robot dynamics
  JerkRate           : REAL;
  /// Index of tool
  /// •      0: Flange (default)
  /// • 1..254: Tool frames
  ToolNo             : USINT;
  /// Index of frame
  /// •      0: WCS (default)
  /// • 1..254: User frames
  FrameNo            : USINT;
  /// Parameter which determines the behavior towards the previously sent and still active or buffered commands
  AbortingMode       : AbortingMode;
  /// Parameter which determines the transition behavior at the end of the movement to be sent to the next command. 
  /// The user can choose a transition type between exact stop and different blend possibilities
  BlendingMode       : BlendingMode;
  /// Additional parameter for the blending mode, to define i.e. velocity limit (%) or blending radius
  BlendingParameter  : ARRAY [0..1] OF REAL := [10,0];
  /// Parameter is used if it is greater than 0 (default)
  /// • Velocity input is ignored
  /// • Parameter defines the time for the movement to reach the target position
  /// Error is sent by the RC if the time cannot be kept
  MoveTime           : TIME;
  /// Parameter to describe how the orientation axes (RX, RY, RZ) will be interpolated during the movement
  OriMode            : OriMode;
  /// Defines the usage of the config byte inside the position according to Table 6-238
  ConfigMode         : ArmConfigParameter;
  /// Defines the usage of the TurnNumber byte inside the position.
  TurnMode           : TurnMode;
  /// Set TRUE to allow manipulation of this move command through superimposing functions.
  /// For more information see chapter 5.5.9.5
  Manipulation       : BOOL;
  /// Defines the target sequence in which the command will be executed
  SequenceFlag       : SequenceFlag;
  /// ID of Action that will be executed when this command is active
  /// • >0: Start Action - Start executing the Action function with the identical ListenerID.
  /// • <0: Stop Action  -  Stop executing the Action function with the identical ListenerID.
  /// • 0: No trigger (default)-  If no EmitterID is defined, the function will not trigger any Action during its execution
  /// For more information see section Triggers of this chapter or chapter 5.5.12.4.
  EmitterID          : ARRAY [0..3] OF SINT;
END_VAR

VAR_OUTPUT
  /// The command has been completed successfully
  Done               : BOOL;
  /// FB is being processed
  Busy               : BOOL;
  /// Command is transferred and confirmed by the RC
  CommandBuffered    : BOOL;
  /// The command takes control of the motion of the according axis group
  Active             : BOOL;
  /// The command was aborted by another command.
  CommandAborted     : BOOL;
  /// TRUE, while command is interrupted during execution and can be continued
  CommandInterrupted : BOOL;
  /// Distance-to-go of the current job.
  /// • -1: No valid value because move command is not yet active (valid values are pending) or not supported by RC
  /// • >0: Actual distance between current and target position
  /// •  0: Target position reached
  RemainingDistance  : REAL;
  /// Percentage of already traversed distance of current job.
  /// If not supported : • -1
  Progress           : REAL;
  /// Unique system-generated ID of the trigger function when the function is called by the user.
  /// For more information see chapter 5.5.12.4.
  FollowID           : DINT;
END_VAR

                  
                

METHOD PROTECTED OnCall
VAR_IN_OUT
  /// Robot assignment of function
  AxesGroup         : AxesGroup; 
END_VAR
                        
                      
END_METHOD
END_FUNCTION_BLOCK

/// Set a trigger in a defined position of a circular path.
FUNCTION_BLOCK MoveCircularCamFB EXTENDS RobotLibraryBaseFB
// ------------------------------------------------------------------------- 
//  SRCI Robot Library                                                
// ------------------------------------------------------------------------- 
//                                                                           
//  Object:      MoveCircularCamFB                                       
//  Author:      Thorsten Brach                                                
//  Date:        2024-06-01
//
//  Description:                                              
//   
//                                                                           
//  Copyright: 
//    (C) 2024 Thorsten Brach. All rights reserved                                                                         
//                                                                           
//  Disclaimer:                                                                           
//    This project is provided without any guarantee and can be used for   
//    private and commercial purposes. Any commercial use is at the user’s 
//    own risk and responsibility.
//
// -------------------------------------------------------------------------
VAR_INPUT
  /// Start of the command at the rising edge
  Execute            : BOOL;
  /// Specifies the meaning of the input parameter "AuxPoint".
  CircMode           : CircMode;
  /// Auxiliary position of the robot in the specified coordinate system, used in for the circle path calculation.
  AuxPoint           : RobotCartesianPosition;
  /// Specifies the circle’s plane when CircMode = 2 is selected
  CircPlane          : CircPlane;
  /// Relates to CircMode =1:
  /// Permissible deviation of the distances from starting point to center point, from auxiliary point to center point and from end point to center point.
  /// These distances must be identical to travel a circular path. When the distance from a point to the center point is within the allowed deviation, 
  /// the position of the center point is adjusted to the mean internally. If the deviation is greater than the specified Tolerance, 
  /// the command returns an error. See also Figure 6-106.
  Tolerance          : REAL;
  /// Absolute end position of the robot in the specified coordinate system. If "CircMode" = 2 this position is ignored 
  EndPoint           : RobotCartesianPosition;
  /// Angle is only used when "CircMode" = 2. 
  /// The circular angle defines the end position of the circular motion. The circular path is defined by the angle, 
  /// the center point ("AuxPoint") and the actual position. Always positive
  Angle              : REAL;
  /// Choice of the path
  PathChoice         : PathChoice;  
  /// TCP velocity in % of nominal velocity
  /// •  <0%: (default) - Use default velocity
  /// •   0%:           - Use internal minimal velocity
  /// • 100%:           - Use maximal reference velocity
  /// See chapter 5.5.7 Robot dynamics
  VelocityRate       : REAL;
  /// Acceleration for movement in % of nominal acceleration
  /// •  <0%: (default) - Use default acceleration
  /// •   0%:           - Use internal minimal acceleration
  /// • 100%:           - Use maximal reference acceleration
  /// See chapter 5.5.7 Robot dynamics
  AccelerationRate   : REAL;
  /// Deceleration for movement in % of nominal deceleration
  /// •  <0%: (default) - Use default deceleration 
  /// •   0%:           - Use internal minimal deceleration
  /// • 100%:           - Use maximal reference deceleration
  /// See chapter 5.5.7 Robot dynamics
  DecelerationRate   : REAL;
  /// Jerk of the movement in % of nominal jerk
  /// •  <0%: (default) - Use default jerk
  /// •   0%:           - Use internal minimal jerk
  /// • 100%:           - Use maximal reference jerk
  /// See chapter 5.5.7 Robot dynamics
  JerkRate           : REAL;
  /// Index of tool
  /// •      0: Flange (default)
  /// • 1..254: Tool frames
  ToolNo             : USINT;
  /// Index of frame
  /// •      0: WCS (default)
  /// • 1..254: User frames
  FrameNo            : USINT;
  /// Parameter which determines the behavior towards the previously sent and still active or buffered commands
  AbortingMode       : AbortingMode;
  /// Parameter which determines the transition behavior at the end of the movement to be sent to the next command. 
  /// The user can choose a transition type between exact stop and different blend possibilities
  BlendingMode       : BlendingMode;
  /// Additional parameter for the blending mode, to define i.e. velocity limit (%) or blending radius
  BlendingParameter  : ARRAY [0..1] OF REAL := [10,0];
  /// Parameter is used if it is greater than 0 (default)
  /// • Velocity input is ignored
  /// • Parameter defines the time for the movement to reach the target position
  /// Error is sent by the RC if the time cannot be kept
  MoveTime           : TIME;
  /// Parameter to describe how the orientation axes (RX, RY, RZ) will be interpolated during the movement
  OriMode            : OriMode;
  /// Defines the usage of the config byte inside the position according to Table 6-238
  ConfigMode         : ArmConfigParameter;
  /// Defines the usage of the TurnNumber byte inside the position.
  TurnMode           : TurnMode;
  /// Specifies the desired byte address that shall be written
  Index              : USINT;
  /// Specifies which output may be written
  OutputBitmask      : BYTE;
  /// Value of Digital Output
  Value              : BYTE;
  /// Reference position for the trigger point (at least one option must be supported):
  /// • 0: Start position (default) O
  /// • 1: End position
  RelativePosition   : BOOL;
  /// Time delay [ms] for the trigger point
  TriggerDelay       : UINT;
  /// Offset in percentage of the movement towards the trigger point in relation to the reference position
  TriggerDistance    : REAL;
  /// Set TRUE to allow manipulation of this move command through superimposing functions.
  /// For more information see chapter 5.5.9.5  
  Manipulation       : BOOL;
  /// Defines the target sequence in which the command will be executed
  SequenceFlag       : SequenceFlag;
END_VAR

VAR_OUTPUT
  /// The command has been completed successfully
  Done               : BOOL;
  /// FB is being processed
  Busy               : BOOL;
  /// Command is transferred and confirmed by the RC
  CommandBuffered    : BOOL;
  /// The command takes control of the motion of the according axis group
  Active             : BOOL;
  /// The command was aborted by another command.
  CommandAborted     : BOOL;
  /// TRUE, while command is interrupted during execution and can be continued
  CommandInterrupted : BOOL;
  /// Distance-to-go of the current job.
  /// • -1: No valid value because move command is not yet active (valid values are pending) or not supported by RC
  /// • >0: Actual distance between current and target position
  /// •  0: Target position reached
  RemainingDistance  : REAL;
  /// Percentage of already traversed distance of current job.
  /// If not supported : • -1
  Progress           : REAL;
END_VAR

                  
                

METHOD PROTECTED OnCall
VAR_IN_OUT
  /// Robot assignment of function
  AxesGroup         : AxesGroup; 
END_VAR
                        
                      
END_METHOD
END_FUNCTION_BLOCK

/// Move the TCP relative to the actual cartesian position (circular interpolation) 
FUNCTION_BLOCK MoveCircularRelativeFB EXTENDS RobotLibraryBaseFB
// ------------------------------------------------------------------------- 
//  SRCI Robot Library                                                
// ------------------------------------------------------------------------- 
//                                                                           
//  Object:      MoveCircularRelativeFB                                       
//  Author:      Thorsten Brach                                                
//  Date:        2024-06-01
//
//  Description:                                              
//   
//                                                                           
//  Copyright: 
//    (C) 2024 Thorsten Brach. All rights reserved                                                                         
//                                                                           
//  Disclaimer:                                                                           
//    This project is provided without any guarantee and can be used for   
//    private and commercial purposes. Any commercial use is at the user’s 
//    own risk and responsibility.
//
// -------------------------------------------------------------------------
VAR_INPUT
  /// Start of the command at the rising edge
  Execute            : BOOL;
  /// Specifies the meaning of the input parameter "AuxPoint".
  CircMode           : CircMode;
  /// Auxiliary position of the robot in the specified coordinate system, used in for the circle path calculation.
  AuxPoint           : RobotCartesianPosition;
  /// Specifies the circle’s plane when CircMode = 2 is selected
  CircPlane          : CircPlane;
  /// Relates to CircMode =1:
  /// Permissible deviation of the distances from starting point to center point, from auxiliary point to center point and from end point to center point.
  /// These distances must be identical to travel a circular path. When the distance from a point to the center point is within the allowed deviation, 
  /// the position of the center point is adjusted to the mean internally. If the deviation is greater than the specified Tolerance, 
  /// the command returns an error. See also Figure 6-106.
  Tolerance          : REAL;
  /// Absolute end position of the robot in the specified coordinate system. If "CircMode" = 2 this position is ignored 
  EndPoint           : RobotCartesianPosition;
  /// Angle is only used when "CircMode" = 2. 
  /// The circular angle defines the end position of the circular motion. The circular path is defined by the angle, 
  /// the center point ("AuxPoint") and the actual position. Always positive
  Angle              : REAL;
  /// Choice of the path
  PathChoice         : PathChoice;  
  /// Defines type of reference coordinate system of the offset position
  ReferenceType      : ReferenceType;
  /// TCP velocity in % of nominal velocity
  /// •  <0%: (default) - Use default velocity
  /// •   0%:           - Use internal minimal velocity
  /// • 100%:           - Use maximal reference velocity
  /// See chapter 5.5.7 Robot dynamics
  VelocityRate       : REAL;
  /// Acceleration for movement in % of nominal acceleration
  /// •  <0%: (default) - Use default acceleration
  /// •   0%:           - Use internal minimal acceleration
  /// • 100%:           - Use maximal reference acceleration
  /// See chapter 5.5.7 Robot dynamics
  AccelerationRate   : REAL;
  /// Deceleration for movement in % of nominal deceleration
  /// •  <0%: (default) - Use default deceleration 
  /// •   0%:           - Use internal minimal deceleration
  /// • 100%:           - Use maximal reference deceleration
  /// See chapter 5.5.7 Robot dynamics
  DecelerationRate   : REAL;
  /// Jerk of the movement in % of nominal jerk
  /// •  <0%: (default) - Use default jerk
  /// •   0%:           - Use internal minimal jerk
  /// • 100%:           - Use maximal reference jerk
  /// See chapter 5.5.7 Robot dynamics
  JerkRate           : REAL;
  /// Index of tool
  /// •      0: Flange (default)
  /// • 1..254: Tool frames
  ToolNo             : USINT;
  /// Index of frame
  /// •      0: WCS (default)
  /// • 1..254: User frames
  FrameNo            : USINT;
  /// Parameter which determines the behavior towards the previously sent and still active or buffered commands
  AbortingMode       : AbortingMode;
  /// Parameter which determines the transition behavior at the end of the movement to be sent to the next command. 
  /// The user can choose a transition type between exact stop and different blend possibilities
  BlendingMode       : BlendingMode;
  /// Additional parameter for the blending mode, to define i.e. velocity limit (%) or blending radius
  BlendingParameter  : ARRAY [0..1] OF REAL := [10,0];
  /// Parameter is used if it is greater than 0 (default)
  /// • Velocity input is ignored
  /// • Parameter defines the time for the movement to reach the target position
  /// Error is sent by the RC if the time cannot be kept
  MoveTime           : TIME;
  /// Parameter to describe how the orientation axes (RX, RY, RZ) will be interpolated during the movement
  OriMode            : OriMode;
  /// Defines the usage of the config byte inside the position according to Table 6-238
  ConfigMode         : ArmConfigParameter;
  /// Defines the usage of the TurnNumber byte inside the position.
  TurnMode           : TurnMode;
  /// Set TRUE to allow manipulation of this move command through superimposing functions.
  /// For more information see chapter 5.5.9.5
  Manipulation       : BOOL;
  /// Defines the target sequence in which the command will be executed
  SequenceFlag       : SequenceFlag;
  /// ID of Action that will be executed when this command is active
  /// • >0: Start Action - Start executing the Action function with the identical ListenerID.
  /// • <0: Stop Action  -  Stop executing the Action function with the identical ListenerID.
  /// • 0: No trigger (default)-  If no EmitterID is defined, the function will not trigger any Action during its execution
  /// For more information see section Triggers of this chapter or chapter 5.5.12.4.
  EmitterID          : ARRAY [0..3] OF SINT;
END_VAR

VAR_OUTPUT
  /// The command has been completed successfully
  Done               : BOOL;
  /// FB is being processed
  Busy               : BOOL;
  /// Command is transferred and confirmed by the RC
  CommandBuffered    : BOOL;
  /// The command takes control of the motion of the according axis group
  Active             : BOOL;
  /// The command was aborted by another command.
  CommandAborted     : BOOL;
  /// TRUE, while command is interrupted during execution and can be continued
  CommandInterrupted : BOOL;
  /// Distance-to-go of the current job.
  /// • -1: No valid value because move command is not yet active (valid values are pending) or not supported by RC
  /// • >0: Actual distance between current and target position
  /// •  0: Target position reached
  RemainingDistance  : REAL;
  /// Percentage of already traversed distance of current job.
  /// If not supported : • -1
  Progress           : REAL;
  /// Unique system-generated ID of the trigger function when the function is called by the user.
  /// For more information see chapter 5.5.12.4.
  FollowID           : DINT;
END_VAR

                  
                

METHOD PROTECTED OnCall
VAR_IN_OUT
  /// Robot assignment of function
  AxesGroup         : AxesGroup; 
END_VAR
                        
                      
END_METHOD
END_FUNCTION_BLOCK

/// Direct Move from actual position to destination through auxiliary
/// position defined by offset in all dimensions (movement to the target position PTP)
FUNCTION_BLOCK MoveDepartDirectFB EXTENDS RobotLibraryBaseFB
// ------------------------------------------------------------------------- 
//  SRCI Robot Library                                                
// ------------------------------------------------------------------------- 
//                                                                           
//  Object:      MoveDepartDirectFB                                       
//  Author:      Thorsten Brach                                                
//  Date:        2024-06-01
//
//  Description:                                              
//   
//                                                                           
//  Copyright: 
//    (C) 2024 Thorsten Brach. All rights reserved                                                                         
//                                                                           
//  Disclaimer:                                                                           
//    This project is provided without any guarantee and can be used for   
//    private and commercial purposes. Any commercial use is at the user’s 
//    own risk and responsibility.
//
// -------------------------------------------------------------------------
VAR_INPUT
  /// Start of the command at the rising edge
  Execute            : BOOL;
  /// Absolute target coordinates in the selected coordinate system (see input parameters ToolNo and FrameNo).
  TargetPosition     : RobotCartesianPosition;
  /// Offset distance of auxiliary position from TargetPosition
  Offset             : AuxOffset;
  /// Defines type of reference coordinate system of the offset position
  ReferenceType      : ReferenceType;
  /// TCP velocity in % of nominal velocity
  /// •  <0%: (default) - Use default velocity
  /// •   0%:           - Use internal minimal velocity
  /// • 100%:           - Use maximal reference velocity
  /// See chapter 5.5.7 Robot dynamics
  VelocityRate       : REAL;
  /// Acceleration for movement in % of nominal acceleration
  /// •  <0%: (default) - Use default acceleration
  /// •   0%:           - Use internal minimal acceleration
  /// • 100%:           - Use maximal reference acceleration
  /// See chapter 5.5.7 Robot dynamics
  AccelerationRate   : REAL;
  /// Deceleration for movement in % of nominal deceleration
  /// •  <0%: (default) - Use default deceleration 
  /// •   0%:           - Use internal minimal deceleration
  /// • 100%:           - Use maximal reference deceleration
  /// See chapter 5.5.7 Robot dynamics
  DecelerationRate   : REAL;
  /// Jerk of the movement in % of nominal jerk
  /// •  <0%: (default) - Use default jerk
  /// •   0%:           - Use internal minimal jerk
  /// • 100%:           - Use maximal reference jerk
  /// See chapter 5.5.7 Robot dynamics
  JerkRate           : REAL;
  /// Index of tool
  /// •      0: Flange (default)
  /// • 1..254: Tool frames
  ToolNo             : USINT;
  /// Index of frame
  /// •      0: WCS (default)
  /// • 1..254: User frames
  FrameNo            : USINT;
  /// Parameter which determines the behavior towards the previously sent and still active or buffered commands
  AbortingMode       : AbortingMode;
  /// Parameter which determines the transition behavior at the end of the movement to be sent to the next command. 
  /// The user can choose a transition type between exact stop and different blend possibilities
  BlendingMode       : BlendingMode;
  /// Additional parameter for the blending mode, to define i.e. velocity limit (%) or blending radius
  BlendingParameter  : ARRAY [0..1] OF REAL := [10,0];
  /// Define blending sphere with radius around auxiliary position. For exact stop define AuxCornerDistance = 0
  AuxCornerDistance  : REAL;
  /// Parameter is used if it is greater than 0 (default)
  /// • Velocity input is ignored
  /// • Parameter defines the time for the movement to reach the target position
  /// Error is sent by the RC if the time cannot be kept
  MoveTime           : TIME;
  /// Parameter to describe how the orientation axes (RX, RY, RZ) will be interpolated during the movement
  OriMode            : OriMode;
  /// Defines the usage of the config byte inside the position according to Table 6-238
  ConfigMode         : ArmConfigParameter;
  /// Defines the usage of the TurnNumber byte inside the position.
  TurnMode           : TurnMode;
  /// Factor by which VelocityRate is multiplied to define the velocity for the second segment of the motion. Always positive.
  /// • 0: use the minimal velocity
  /// • 1: use the velocity set with VelocityRate 
  /// Input values below 1 to reduce velocity, 
  /// Input values above 1 to increase velocity.
  /// See chapter 5.5.7 Robot dynamics
  VelocityCoefficient: REAL;
  /// Set TRUE to allow manipulation of this move command through superimposing functions.
  /// For more information see chapter 5.5.9.5
  Manipulation       : BOOL;
  /// Defines the target sequence in which the command will be executed
  SequenceFlag       : SequenceFlag;
  /// ID of Action that will be executed when this command is active
  /// • >0: Start Action - Start executing the Action function with the identical ListenerID.
  /// • <0: Stop Action  -  Stop executing the Action function with the identical ListenerID.
  /// • 0: No trigger (default)-  If no EmitterID is defined, the function will not trigger any Action during its execution
  /// For more information see section Triggers of this chapter or chapter 5.5.12.4.
  EmitterID          : ARRAY [0..3] OF SINT;
END_VAR

VAR_OUTPUT
  /// The command has been completed successfully
  Done               : BOOL;
  /// FB is being processed
  Busy               : BOOL;
  /// Command is transferred and confirmed by the RC
  CommandBuffered    : BOOL;
  /// The command takes control of the motion of the according axis group
  Active             : BOOL;
  /// The command was aborted by another command.
  CommandAborted     : BOOL;
  /// TRUE, while command is interrupted during execution and can be continued
  CommandInterrupted : BOOL;
  /// Distance-to-go of the current job.
  /// • -1: No valid value because move command is not yet active (valid values are pending) or not supported by RC
  /// • >0: Actual distance between current and target position
  /// •  0: Target position reached
  RemainingDistance  : REAL;
  /// Percentage of already traversed distance of current job.
  /// If not supported : • -1
  Progress           : REAL;
  /// Unique system-generated ID of the trigger function when the function is called by the user.
  /// For more information see chapter 5.5.12.4.
  FollowID           : DINT;
END_VAR

                  
                

METHOD PROTECTED OnCall
VAR_IN_OUT
  /// Robot assignment of function
  AxesGroup         : AxesGroup; 
END_VAR
                        
                      
END_METHOD
END_FUNCTION_BLOCK

/// Linear Move from actual position to destination through auxiliary position,
/// defined by offset in all dimensions (movement to target position linear)
FUNCTION_BLOCK MoveDepartLinearFB EXTENDS RobotLibraryBaseFB
// ------------------------------------------------------------------------- 
//  SRCI Robot Library                                                
// ------------------------------------------------------------------------- 
//                                                                           
//  Object:      MoveDepartLinearFB                                       
//  Author:      Thorsten Brach                                                
//  Date:        2024-06-01
//
//  Description:                                              
//   
//                                                                           
//  Copyright: 
//    (C) 2024 Thorsten Brach. All rights reserved                                                                         
//                                                                           
//  Disclaimer:                                                                           
//    This project is provided without any guarantee and can be used for   
//    private and commercial purposes. Any commercial use is at the user’s 
//    own risk and responsibility.
//
// -------------------------------------------------------------------------
VAR_INPUT
  /// Start of the command at the rising edge
  Execute            : BOOL;
  /// Absolute target coordinates in the selected coordinate system (see input parameters ToolNo and FrameNo).
  TargetPosition     : RobotCartesianPosition;
  /// Offset distance of auxiliary position from TargetPosition
  Offset             : AuxOffset;
  /// Defines type of reference coordinate system of the offset position
  ReferenceType      : ReferenceType;
  /// TCP velocity in % of nominal velocity
  /// •  <0%: (default) - Use default velocity
  /// •   0%:           - Use internal minimal velocity
  /// • 100%:           - Use maximal reference velocity
  /// See chapter 5.5.7 Robot dynamics
  VelocityRate       : REAL;
  /// Acceleration for movement in % of nominal acceleration
  /// •  <0%: (default) - Use default acceleration
  /// •   0%:           - Use internal minimal acceleration
  /// • 100%:           - Use maximal reference acceleration
  /// See chapter 5.5.7 Robot dynamics
  AccelerationRate   : REAL;
  /// Deceleration for movement in % of nominal deceleration
  /// •  <0%: (default) - Use default deceleration 
  /// •   0%:           - Use internal minimal deceleration
  /// • 100%:           - Use maximal reference deceleration
  /// See chapter 5.5.7 Robot dynamics
  DecelerationRate   : REAL;
  /// Jerk of the movement in % of nominal jerk
  /// •  <0%: (default) - Use default jerk
  /// •   0%:           - Use internal minimal jerk
  /// • 100%:           - Use maximal reference jerk
  /// See chapter 5.5.7 Robot dynamics
  JerkRate           : REAL;
  /// Index of tool
  /// •      0: Flange (default)
  /// • 1..254: Tool frames
  ToolNo             : USINT;
  /// Index of frame
  /// •      0: WCS (default)
  /// • 1..254: User frames
  FrameNo            : USINT;
  /// Parameter which determines the behavior towards the previously sent and still active or buffered commands
  AbortingMode       : AbortingMode;
  /// Parameter which determines the transition behavior at the end of the movement to be sent to the next command. 
  /// The user can choose a transition type between exact stop and different blend possibilities
  BlendingMode       : BlendingMode;
  /// Additional parameter for the blending mode, to define i.e. velocity limit (%) or blending radius
  BlendingParameter  : ARRAY [0..1] OF REAL := [10,0];
  /// Define blending sphere with radius around auxiliary position. For exact stop define AuxCornerDistance = 0
  AuxCornerDistance  : REAL;
  /// Parameter is used if it is greater than 0 (default)
  /// • Velocity input is ignored
  /// • Parameter defines the time for the movement to reach the target position
  /// Error is sent by the RC if the time cannot be kept
  MoveTime           : TIME;
  /// Parameter to describe how the orientation axes (RX, RY, RZ) will be interpolated during the movement
  OriMode            : OriMode;
  /// Defines the usage of the config byte inside the position according to Table 6-238
  ConfigMode         : ArmConfigParameter;
  /// Defines the usage of the TurnNumber byte inside the position.
  TurnMode           : TurnMode;
  /// Factor by which VelocityRate is multiplied to define the velocity for the second segment of the motion. Always positive.
  /// • 0: use the minimal velocity
  /// • 1: use the velocity set with VelocityRate 
  /// Input values below 1 to reduce velocity, 
  /// Input values above 1 to increase velocity.
  /// See chapter 5.5.7 Robot dynamics
  VelocityCoefficient: REAL;
  /// Set TRUE to allow manipulation of this move command through superimposing functions.
  /// For more information see chapter 5.5.9.5
  Manipulation       : BOOL;
  /// Defines the target sequence in which the command will be executed
  SequenceFlag       : SequenceFlag;
  /// ID of Action that will be executed when this command is active
  /// • >0: Start Action - Start executing the Action function with the identical ListenerID.
  /// • <0: Stop Action  -  Stop executing the Action function with the identical ListenerID.
  /// • 0: No trigger (default)-  If no EmitterID is defined, the function will not trigger any Action during its execution
  /// For more information see section Triggers of this chapter or chapter 5.5.12.4.
  EmitterID          : ARRAY [0..3] OF SINT;
END_VAR

VAR_OUTPUT
  /// The command has been completed successfully
  Done               : BOOL;
  /// FB is being processed
  Busy               : BOOL;
  /// Command is transferred and confirmed by the RC
  CommandBuffered    : BOOL;
  /// The command takes control of the motion of the according axis group
  Active             : BOOL;
  /// The command was aborted by another command.
  CommandAborted     : BOOL;
  /// TRUE, while command is interrupted during execution and can be continued
  CommandInterrupted : BOOL;
  /// Distance-to-go of the current job.
  /// • -1: No valid value because move command is not yet active (valid values are pending) or not supported by RC
  /// • >0: Actual distance between current and target position
  /// •  0: Target position reached
  RemainingDistance  : REAL;
  /// Percentage of already traversed distance of current job.
  /// If not supported : • -1
  Progress           : REAL;
  /// Unique system-generated ID of the trigger function when the function is called by the user.
  /// For more information see chapter 5.5.12.4.
  FollowID           : DINT;
END_VAR

                  
                

METHOD PROTECTED OnCall
VAR_IN_OUT
  /// Robot assignment of function
  AxesGroup         : AxesGroup; 
END_VAR
                        
                      
END_METHOD
END_FUNCTION_BLOCK

/// Move Joints to an absolute cartesian position (Absolute cartesian PTP) (Joint interpolated movement)
FUNCTION_BLOCK MoveDirectAbsoluteFB EXTENDS RobotLibraryBaseFB
// ------------------------------------------------------------------------- 
//  SRCI Robot Library                                                
// ------------------------------------------------------------------------- 
//                                                                           
//  Object:      MoveDirectAbsoluteFB                                       
//  Author:      Thorsten Brach                                                
//  Date:        2024-06-01
//
//  Description:                                              
//   
//                                                                           
//  Copyright: 
//    (C) 2024 Thorsten Brach. All rights reserved                                                                         
//                                                                           
//  Disclaimer:                                                                           
//    This project is provided without any guarantee and can be used for   
//    private and commercial purposes. Any commercial use is at the user’s 
//    own risk and responsibility.
//
// -------------------------------------------------------------------------
VAR_INPUT
  /// Start of the command at the rising edge
  Execute            : BOOL;
  /// Absolute target coordinates in the selected coordinate system (see input parameters ToolNo and FrameNo)
  Position           : RobotCartesianPosition;
  /// TCP velocity in % of nominal velocity
  /// •  <0%: (default) - Use default velocity
  /// •   0%:           - Use internal minimal velocity
  /// • 100%:           - Use maximal reference velocity
  /// See chapter 5.5.7 Robot dynamics
  VelocityRate       : REAL;
  /// Acceleration for movement in % of nominal acceleration
  /// •  <0%: (default) - Use default acceleration
  /// •   0%:           - Use internal minimal acceleration
  /// • 100%:           - Use maximal reference acceleration
  /// See chapter 5.5.7 Robot dynamics
  AccelerationRate   : REAL;
  /// Deceleration for movement in % of nominal deceleration
  /// •  <0%: (default) - Use default deceleration 
  /// •   0%:           - Use internal minimal deceleration
  /// • 100%:           - Use maximal reference deceleration
  /// See chapter 5.5.7 Robot dynamics
  DecelerationRate   : REAL;
  /// Jerk of the movement in % of nominal jerk
  /// •  <0%: (default) - Use default jerk
  /// •   0%:           - Use internal minimal jerk
  /// • 100%:           - Use maximal reference jerk
  /// See chapter 5.5.7 Robot dynamics
  JerkRate           : REAL;
  /// Index of tool
  /// •      0: Flange (default)
  /// • 1..254: Tool frames
  ToolNo             : USINT;
  /// Index of frame
  /// •      0: WCS (default)
  /// • 1..254: User frames
  FrameNo            : USINT;
  /// Parameter which determines the behavior towards the previously sent and still active or buffered commands
  AbortingMode       : AbortingMode;
  /// Parameter which determines the transition behavior at the end of the movement to be sent to the next command. 
  /// The user can choose a transition type between exact stop and different blend possibilities
  BlendingMode       : BlendingMode;
  /// Additional parameter for the blending mode, to define i.e. velocity limit (%) or blending radius
  BlendingParameter  : ARRAY [0..1] OF REAL := [10,0];
  /// Parameter is used if it is greater than 0 (default)
  /// • Velocity input is ignored
  /// • Parameter defines the time for the movement to reach the target position
  /// Error is sent by the RC if the time cannot be kept
  MoveTime           : TIME;
  /// Defines the usage of the config byte inside the position according to Table 6-238
  ConfigMode         : ArmConfigParameter;
  /// Defines the usage of the TurnNumber byte inside the position.
  TurnMode           : TurnMode;
  /// Set TRUE to allow manipulation of this move command through superimposing functions.
  /// For more information see chapter 5.5.9.5
  Manipulation       : BOOL;
  /// Defines the target sequence in which the command will be executed
  SequenceFlag       : SequenceFlag;
  /// ID of Action that will be executed when this command is active
  /// • >0: Start Action - Start executing the Action function with the identical ListenerID.
  /// • <0: Stop Action  -  Stop executing the Action function with the identical ListenerID.
  /// • 0: No trigger (default)-  If no EmitterID is defined, the function will not trigger any Action during its execution
  /// For more information see section Triggers of this chapter or chapter 5.5.12.4.
  EmitterID          : ARRAY [0..3] OF SINT;
END_VAR

VAR_OUTPUT
  /// The command has been completed successfully
  Done               : BOOL;
  /// FB is being processed
  Busy               : BOOL;
  /// Command is transferred and confirmed by the RC
  CommandBuffered    : BOOL;
  /// The command takes control of the motion of the according axis group
  Active             : BOOL;
  /// The command was aborted by another command.
  CommandAborted     : BOOL;
  /// TRUE, while command is interrupted during execution and can be continued
  CommandInterrupted : BOOL;
  /// Distance-to-go of the current job.
  /// • -1: No valid value because move command is not yet active (valid values are pending) or not supported by RC
  /// • >0: Actual distance between current and target position
  /// •  0: Target position reached
  RemainingDistance  : REAL;
  /// Percentage of already traversed distance of current job.
  /// If not supported : • -1
  Progress           : REAL;
  /// Unique system-generated ID of the trigger function when the function is called by the user.
  /// For more information see chapter 5.5.12.4.
  FollowID           : DINT;
END_VAR

                  
                

METHOD PROTECTED OnCall
VAR_IN_OUT
  /// Robot assignment of function
  AxesGroup         : AxesGroup; 
END_VAR
                        
                      
END_METHOD
END_FUNCTION_BLOCK

